FUNCTION_BLOCK WoodBunkTable EXTENDS MaterialHolder
VAR_OUTPUT
	occupied AT %I* : ARRAY[1..numSlots] OF BOOL; //sensors must turn HIGH before bunk arrives, and turn LOW after bunk leaves
END_VAR
VAR
	i : INT(1..10);
END_VAR
VAR_STAT CONSTANT
	numSlots : INT := 10;
END_VAR

(*
FOR i:=1 TO numSlots BY 1 DO
	IF NOT occupied[i] THEN
		slots[i] := '';
	END_IF
END_FOR
*)

METHOD autofill : BOOL
VAR_INPUT
	materialID : STRING;
END_VAR
VAR
	i : INT;
	slot : INT;
END_VAR
(*
this method will automatically find an open slot
*)
IF isFull() OR materialID = '' THEN
	RETURN;
END_IF

IF findOpenSlot(materialID, openSlot=> slot) THEN
	place(slot, materialID);
	autofill := TRUE;
	
	//ADSLOGSTR(msgCtrlMask := ADSLOG_MSGTYPE_ERROR , msgFmtStr := 'autofill: %s', strArg := materialID);
END_IF
END_METHOD

METHOD findOpenSlot : BOOL
VAR_INPUT
	materialID : STRING;
END_VAR
VAR_OUTPUT
	openSlot : INT := 0;
END_VAR
VAR
	i : INT;
END_VAR
IF FIND(materialID, 'WDW') > 0 THEN //top wide, load in slot 9-10
	FOR i:=9 TO 10 BY 1 DO
		IF slots[i] = '' THEN
			findOpenSlot := TRUE;
			openSlot := i;
			RETURN;
		END_IF
	END_FOR
	
//ELSIF FIND(materialID, 'WDT') > 0 OR FIND(materialID, 'WDS') > 0 THEN //standard width, load in slot 3-10
ELSIF FIND(materialID, 'WD') > 0 THEN //standard width, load in slot 1-8
	FOR i:=1 TO 8 BY 1 DO
		IF slots[i] = '' THEN
			findOpenSlot := TRUE;
			openSlot := i;
			RETURN;
		END_IF
	END_FOR
	
END_IF
END_METHOD

METHOD findSlot : BOOL
VAR_INPUT
	materialID : STRING;
END_VAR
VAR_OUTPUT
	atSlot : INT;
END_VAR
VAR
	i : INT;
END_VAR
FOR i:=1 TO numSlots BY 1 DO
	IF slots[i] = materialID THEN
		atSlot := i;
		findSlot := TRUE;
		RETURN;
	END_IF
END_FOR
END_METHOD

METHOD isEmpty : BOOL
VAR
	i : INT;
	temp : BOOL;
END_VAR
FOR i:=1 TO numSlots BY 1 DO
	temp := temp OR occupied[i]; //TRUE if any slots are occupied
END_FOR

isEmpty := NOT temp; //invert result - FALSE if any slots are occupied
END_METHOD

METHOD isFull : BOOL
VAR
	i : INT;
	temp : BOOL := TRUE;
END_VAR
FOR i:=1 TO numSlots BY 1 DO
	temp := temp AND occupied[i];
END_FOR

isFull := TEMP;
END_METHOD

METHOD place : BOOL
VAR_INPUT
	i : INT;
	materialID : STRING;
END_VAR
IF slots[i] = '' THEN
	slots[i] := materialID;
	place := TRUE;
END_IF
END_METHOD

METHOD remove : BOOL
VAR_INPUT
	i : INT;
END_VAR
VAR_OUTPUT
	materialID : STRING;
END_VAR
remove := slots[i] <> '';

materialID := slots[i];
slots[i] := '';
END_METHOD

END_FUNCTION_BLOCK

(* stored: Version 1.1.0.1, ProductVersion 3.1.4024.11
   POU WoodBunkTable: Id {dc0f3bd0-85c7-41ea-839e-cecdb56a654c}, SpecialFunc None
   Method autofill: Id {0b1558f0-abe0-46a4-ba25-2d74dda1538c}
   Method findOpenSlot: Id {4ad7fd0b-197f-42ee-aa6d-941184505c0d}
   Method findSlot: Id {43e5bcb3-33a4-445d-ab40-bb9cefd27ac2}
   Method isEmpty: Id {a89780a4-d604-444d-ba70-4bd950a2e867}
   Method isFull: Id {a709fd63-7090-49a1-8c6d-2d710e9ddde8}
   Method place: Id {47c85d53-1f37-4db8-9692-6ad12f349b85}
   Method remove: Id {426c1438-d5a3-4715-8770-70aeabf0c7fb} *)
